{attribute 'pack_mode' := '2'}
TYPE ST_MOVER_CTRL :
STRUCT
  Cmd             : E_MOVER_CTRL;  // order to execute on mover
END_STRUCT
END_TYPE

(* stored: Version 1.1.0.1, ProductVersion 3.1.4024.15
   DUT ST_MOVER_CTRL: Id {a299673c-c2cc-439a-8430-207ccf2653ce} *)
